// TIA Portal V17 export
// export: Created 2025-03-07T09:24:10.8160343Z, ExportSetting WithDefaults, DisplayName Totally Integrated Automation Portal, DisplayVersion V17 Update 8, DisplayName TIA Portal Openness, DisplayVersion V17 Update 8, DisplayName TIA Portal Version Control Interface, DisplayVersion V17, DisplayName SINAMICS Startdrive Advanced, DisplayVersion V17 SP2, DisplayName SINAMICS Startdrive G110M, G120, G120C, G120D, G120P, G115D, DisplayVersion V17 SP2, DisplayName SINAMICS Startdrive G130, G150, S120, S150, SINAMICS MV, S210, DisplayVersion V17 SP2, DisplayName STEP 7 Professional, DisplayVersion V17 Update 8, DisplayName SINUMERIK ONE STEP 7 Toolbox, DisplayVersion V17 Update 12, DisplayName SINUMERIK 840D sl STEP 7 Toolbox, DisplayVersion V17 Update 12, DisplayName STEP 7 Safety, DisplayVersion V17 Update 6, DisplayName WinCC Advanced, DisplayVersion V17 Update 8
DATA_BLOCK "DB22105_HIGH_LEVEL_HOPPER_1_UNIT_01"   // DB22105
{ DB_Accessible_From_OPC_UA := 'FALSE' }
VERSION : 0.1
// stored: AutoNumber false, DBAccessibleFromOPCUA false, DBAccessibleFromWebserver true, InstanceOfName FB22103_POWDER_LEVEL_SENSOR, InstanceOfType FB
"FB22103_POWDER_LEVEL_SENSOR"
   // VAR_INPUT
   //    iLOW_LEVEL_SENSOR : Bool;
   //    iHIGH_LEVEL_SENSOR : Bool;
   //    iCLEAR_LOG : Bool;
   // END_VAR
   // VAR_OUTPUT
   //    oLOW_LEVEL_WRN : Bool;
   //    "oHIGH LEVEL_WRN" : Bool;
   // END_VAR
   // VAR RETAIN
   //    OUTPUT : Struct
   //       DIGITAL_OUTPUT : Bool;
   //    END_STRUCT;
   //    INPUT_SETINGS : Struct
   //       UNIT_NUMBER : Int;
   //       HOPPER_NUMBER : Int;
   //    END_STRUCT;
   //    ALARMS : Struct
   //       SENSOR_DISCORDANCY_ALM : Bool;
   //    END_STRUCT;
   //    LOG : Struct
   //       LAST_EDGE_LOW_LVL : Date_And_Time;
   //       LAST_EDGE_HIGH_LVL : Date_And_Time;
   //    END_STRUCT;
   //    INTERNAL : Struct
   //       RET_VAL : Int;
   //       AUX1 : Bool;
   //       AUX2 : Bool;
   //    END_STRUCT;
   // END_VAR
BEGIN
END_DATA_BLOCK
